// TIA Portal V17 export
// export: Created 2025-03-07T09:19:14.8092135Z, ExportSetting WithDefaults, DisplayName Totally Integrated Automation Portal, DisplayVersion V17 Update 8, DisplayName TIA Portal Openness, DisplayVersion V17 Update 8, DisplayName TIA Portal Version Control Interface, DisplayVersion V17, DisplayName SINAMICS Startdrive Advanced, DisplayVersion V17 SP2, DisplayName SINAMICS Startdrive G110M, G120, G120C, G120D, G120P, G115D, DisplayVersion V17 SP2, DisplayName SINAMICS Startdrive G130, G150, S120, S150, SINAMICS MV, S210, DisplayVersion V17 SP2, DisplayName STEP 7 Professional, DisplayVersion V17 Update 8, DisplayName SINUMERIK ONE STEP 7 Toolbox, DisplayVersion V17 Update 12, DisplayName SINUMERIK 840D sl STEP 7 Toolbox, DisplayVersion V17 Update 12, DisplayName STEP 7 Safety, DisplayVersion V17 Update 6, DisplayName WinCC Advanced, DisplayVersion V17 Update 8
DATA_BLOCK "DB7237_IDS_AND_PASSWORDS"   // DB7237
{ S7_Optimized_Access := 'FALSE'; DB_Accessible_From_OPC_UA := 'FALSE' }
AUTHOR : ETXETAR
VERSION : 1.0
// stored: AutoNumber false, DBAccessibleFromOPCUA false, DBAccessibleFromWebserver true, IsOnlyStoredInLoadMemory false, IsWriteProtectedInAS false
   VAR RETAIN
      ANY_ID_OK : Bool;   // ANY ID OK
      ANY_PASSWORD_OK : Bool;   // ANY PASSWORD OK
      RESET_PASSWORD : Bool;   // RESET PASSWORD
      RESET_PASSWORD_AUX : Bool;   // RESET PASSWORD AUXILIARY
      AUX_TIMER_RESET : Bool;   // TIMER RESET AUXILIARY
      SCREEN_ID_1 : Byte;   // SCREEN ID 1
      SCREEN_ID_2 : Byte;   // SCREEN ID 2
      SCREEN_AUX : Int;   // SCREEN AUXILIARY
      HMI_USER_ID : Array[1..10] of Char;   // HMI USER ID
      HMI_PASSWORD : Array[1..10] of Char;   // HMI PASSWORD
      HMI_USER_ID_HISTORY : Array[1..10] of Char;   // HMI USER ID HISTORY
      HMI_PASSWORD_HISTORY : Array[1..10] of Char;   // HMI PASSWORD HISTORY
      USER_ID_1 : Array[1..10] of Char;   // HMI USER ID 1
      USER_ID_2 : Array[1..10] of Char;   // HMI USER ID 2
      USER_ID_3 : Array[1..10] of Char;   // HMI USER ID 3
      USER_ID_4 : Array[1..10] of Char;   // HMI USER ID 4
      USER_ID_5 : Array[1..10] of Char;   // HMI USER ID 5
      PASSWORD_1 : Array[1..10] of Char;   // HMI PASSWORD 1
      PASSWORD_2 : Array[1..10] of Char;   // HMI PASSWORD 2
      PASSWORD_3 : Array[1..10] of Char;   // HMI PASSWORD 3
      PASSWORD_4 : Array[1..10] of Char;   // HMI PASSWORD 4
      PASSWORD_5 : Array[1..10] of Char;   // HMI PASSWORD 5
      ID_OK : Array[1..5] of Bool;   // ID OK
      PASSWORD_OK : Array[1..5] of Bool;   // PASSWORD OK
      TIMER_RESET_PASSWORD_DELAY : TON_TIME;   // RESET PASSWORD DELAY TIMER
      TIMER_RESET_PASSWORD { S7_SetPoint := 'True'} : TON_TIME;   // RESET PASSWORD TIMER
   END_VAR
BEGIN
   HMI_USER_ID[1] := 'U';
   HMI_USER_ID[2] := 'S';
   HMI_USER_ID[3] := 'U';
   HMI_USER_ID[4] := 'A';
   HMI_USER_ID[5] := 'R';
   HMI_USER_ID[6] := 'I';
   HMI_USER_ID[7] := 'O';
   HMI_USER_ID[8] := 'S';
   HMI_PASSWORD[1] := 'P';
   HMI_PASSWORD[2] := 'A';
   HMI_PASSWORD[3..4] := 'S';
   HMI_PASSWORD[5] := 'W';
   HMI_PASSWORD[6] := 'O';
   HMI_PASSWORD[7] := 'R';
   HMI_PASSWORD[8] := 'D';
   USER_ID_1[1] := 'E';
   USER_ID_1[2] := 'T';
   USER_ID_1[3] := 'X';
   USER_ID_1[4] := 'E';
   USER_ID_1[5] := 'T';
   USER_ID_1[6] := 'A';
   USER_ID_1[7] := 'R';
   USER_ID_1[8..10] := '$00';
   USER_ID_2[1] := 'R';
   USER_ID_2[2] := 'E';
   USER_ID_2[3] := 'N';
   USER_ID_2[4] := 'A';
   USER_ID_2[5] := 'U';
   USER_ID_2[6] := 'L';
   USER_ID_2[7] := 'T';
   USER_ID_2[8..10] := '$00';
   USER_ID_3[1] := 'O';
   USER_ID_3[2] := 'P';
   USER_ID_3[3] := 'E';
   USER_ID_3[4] := 'R';
   USER_ID_3[5] := 'A';
   USER_ID_3[6] := 'T';
   USER_ID_3[7] := 'O';
   USER_ID_3[8] := 'R';
   USER_ID_3[9..10] := '$00';
   USER_ID_4[1] := 'E';
   USER_ID_4[2] := 'T';
   USER_ID_4[3] := 'X';
   USER_ID_4[4] := 'E';
   USER_ID_4[5] := 'T';
   USER_ID_4[6] := 'A';
   USER_ID_4[7] := 'R';
   USER_ID_4[8] := '1';
   USER_ID_4[9..10] := '$00';
   USER_ID_5[1] := 'E';
   USER_ID_5[2] := 'T';
   USER_ID_5[3] := 'X';
   USER_ID_5[4] := 'E';
   USER_ID_5[5] := 'T';
   USER_ID_5[6] := 'A';
   USER_ID_5[7] := 'R';
   USER_ID_5[8] := '2';
   USER_ID_5[9..10] := '$00';
   PASSWORD_1[1] := '1';
   PASSWORD_1[2] := '2';
   PASSWORD_1[3] := '3';
   PASSWORD_1[4] := '4';
   PASSWORD_1[5] := '5';
   PASSWORD_1[6] := 'A';
   PASSWORD_1[7] := 'B';
   PASSWORD_1[8] := 'C';
   PASSWORD_1[9] := 'D';
   PASSWORD_1[10] := 'E';
   PASSWORD_2[1] := 'M';
   PASSWORD_2[2] := 'A';
   PASSWORD_2[3] := 'I';
   PASSWORD_2[4] := 'N';
   PASSWORD_2[5] := 'T';
   PASSWORD_2[6..10] := '$00';
   PASSWORD_3[1] := 'O';
   PASSWORD_3[2] := 'P';
   PASSWORD_3[3] := 'E';
   PASSWORD_3[4] := 'R';
   PASSWORD_3[5] := 'A';
   PASSWORD_3[6] := 'T';
   PASSWORD_3[7] := 'O';
   PASSWORD_3[8] := 'R';
   PASSWORD_3[9..10] := '$00';
   PASSWORD_4[1] := '1';
   PASSWORD_4[2] := '2';
   PASSWORD_4[3] := '3';
   PASSWORD_4[4] := '4';
   PASSWORD_4[5] := '5';
   PASSWORD_4[6] := 'A';
   PASSWORD_4[7] := 'B';
   PASSWORD_4[8] := 'C';
   PASSWORD_4[9] := 'D';
   PASSWORD_4[10] := 'E';
   PASSWORD_5[1] := '1';
   PASSWORD_5[2] := '2';
   PASSWORD_5[3] := '3';
   PASSWORD_5[4] := '4';
   PASSWORD_5[5] := '5';
   PASSWORD_5[6] := 'A';
   PASSWORD_5[7] := 'B';
   PASSWORD_5[8] := 'C';
   PASSWORD_5[9] := 'D';
   PASSWORD_5[10] := 'E';
   TIMER_RESET_PASSWORD_DELAY.PT := T#2s;
   TIMER_RESET_PASSWORD.PT := T#10M;
END_DATA_BLOCK
